// TIA Portal V17 export
// export: Created 2025-08-05T09:35:59.5209071Z, ExportSetting WithDefaults, DisplayName Totally Integrated Automation Portal, DisplayVersion V17, DisplayName TIA Portal Openness, DisplayVersion V17, DisplayName TIA Portal Version Control Interface, DisplayVersion V17, DisplayName SINAMICS Startdrive Advanced, DisplayVersion V17, DisplayName SINAMICS Startdrive G130, G150, S120, S150, SINAMICS MV, S210, DisplayVersion V17, DisplayName SINAMICS Startdrive G110M, G120, G120C, G120D, G120P, G115D, DisplayVersion V17, DisplayName STEP 7 Professional, DisplayVersion V17, DisplayName STEP 7 Safety, DisplayVersion V17, DisplayName WinCC Advanced, DisplayVersion V17
TYPE "typeFgControlGeneral"
TITLE = Control interface / Steuershnittstelle
// Control interface [V 01.02 | Kernel_V2] / Steuershnittstelle [V 01.02 | Kernel_V2]
// stored: IsFailsafeCompliant false
   STRUCT
      homePosConditions : Bool;   // Grundstellungsbedingungen / Home position conditions
      waitingPositionStep : Bool;   // Warteschritt / Waiting step
      homePostionStep : Bool := TRUE;   // Grundstellungsschritt akitv / Home position step active
      withoutExecutionStep : Bool;   // Schritt ohne Bewegung / Step without movement
      jobNumber : Int;   // Auftragsnummer / Job number
      activeJobNumber : Int := -1;   // Aktive Auftragsnummer von Ablaufsteuerung / Active job number from sequence control
      seqNumber : Int;   // Schrittnummer / Step number
      internalSignals : Struct   // Steuersignale (nur für internen gebrauch!) ... / Control signals (for internal use only!) ...
         startDelayed : Struct   // Verzögerte Startsingale... / Delayed start signals...
            inExecution : Bool;   // Start aktiv verzögert / Start active delayed
            inExecutionPulse : Bool;   // Start aktiv Impuls verzögert / Start active impulse delayed
         END_STRUCT;
      END_STRUCT;
   END_STRUCT;
END_TYPE
